(* IEC 61131-3 sources: ecmc_plugin_strucpp/examples/psi_ioc_examples/MTEST04-MTN-STRUCPP/src/generated, 1 file *)

(* ---- main_bundle.st ---- *)
(* Auto-generated by strucpp_bundle_st.py. *)

(* BEGIN ecmc_control.st *)
FUNCTION_BLOCK ECMC_PID
VAR_INPUT
  Enable   : BOOL := TRUE;
  Reset    : BOOL := FALSE;
  Setpoint : LREAL;
  Actual   : LREAL;
  FF       : LREAL := 0.0;
  Kp       : LREAL := 1.0;
  Ki       : LREAL := 0.0;
  Kd       : LREAL := 0.0;
  Kff      : LREAL := 1.0;
  DT       : LREAL := 1.0;
  DFilterTau : LREAL := 0.0;
  OutMin   : LREAL := 0.0;
  OutMax   : LREAL := 0.0;
  IMin     : LREAL := 0.0;
  IMax     : LREAL := 0.0;
END_VAR
VAR_OUTPUT
  Error   : LREAL;
  Output  : LREAL;
  PPart   : LREAL;
  IPart   : LREAL;
  DPart   : LREAL;
  FFPart  : LREAL;
  Limited : BOOL;
END_VAR
VAR
  PrevError    : LREAL;
  DState       : LREAL;
  WasEnabled   : BOOL;
  CandidateI   : LREAL;
  DRaw         : LREAL;
  DAlpha       : LREAL;
  UnsatOutput  : LREAL;
END_VAR

Error := Setpoint - Actual;

IF Reset THEN
  Output := 0.0;
  PPart := 0.0;
  IPart := 0.0;
  DPart := 0.0;
  FFPart := 0.0;
  Limited := FALSE;
  PrevError := Error;
  DState := 0.0;
  WasEnabled := FALSE;
ELSIF NOT Enable THEN
  Error := Setpoint - Actual;
  Output := 0.0;
  PPart := 0.0;
  DPart := 0.0;
  FFPart := FF * Kff;
  Limited := FALSE;
  PrevError := Error;
  DState := 0.0;
  WasEnabled := FALSE;
ELSIF NOT WasEnabled THEN
  PPart := Error * Kp;
  DPart := 0.0;
  FFPart := FF * Kff;
  UnsatOutput := PPart + IPart + FFPart;
  Output := UnsatOutput;
  Limited := FALSE;

  IF OutMax > OutMin THEN
    IF Output > OutMax THEN
      Output := OutMax;
      Limited := TRUE;
    END_IF;
    IF Output < OutMin THEN
      Output := OutMin;
      Limited := TRUE;
    END_IF;
  END_IF;

  PrevError := Error;
  DState := 0.0;
  WasEnabled := TRUE;
ELSE
  PPart := Error * Kp;
  CandidateI := IPart + Error * Ki * DT;

  IF IMax > IMin THEN
    IF CandidateI > IMax THEN
      CandidateI := IMax;
    END_IF;
    IF CandidateI < IMin THEN
      CandidateI := IMin;
    END_IF;
  END_IF;

  IF DT > 0.0 THEN
    DRaw := (Error - PrevError) / DT;
    IF DFilterTau > 0.0 THEN
      DAlpha := DT / (DFilterTau + DT);
      DState := DState + DAlpha * (DRaw - DState);
    ELSE
      DState := DRaw;
    END_IF;
    DPart := Kd * DState;
  ELSE
    DState := 0.0;
    DPart := 0.0;
  END_IF;

  FFPart := FF * Kff;
  UnsatOutput := PPart + CandidateI + DPart + FFPart;
  Output := UnsatOutput;
  Limited := FALSE;

  IF OutMax > OutMin THEN
    IF Output > OutMax THEN
      Output := OutMax;
      Limited := TRUE;
    END_IF;
    IF Output < OutMin THEN
      Output := OutMin;
      Limited := TRUE;
    END_IF;
  END_IF;

  IF (NOT Limited) OR
     ((UnsatOutput > OutMax) AND (Error < 0.0)) OR
     ((UnsatOutput < OutMin) AND (Error > 0.0)) THEN
    IPart := CandidateI;
  END_IF;

  PrevError := Error;
  WasEnabled := TRUE;
END_IF;
END_FUNCTION_BLOCK
(* END ecmc_control.st *)

(* BEGIN ecmc_utils.st *)
FUNCTION_BLOCK ECMC_DebounceBool
VAR_INPUT
  In       : BOOL;
  OnDelay  : TIME := T#0ms;
  OffDelay : TIME := T#0ms;
END_VAR
VAR_OUTPUT
  Out     : BOOL;
  Rising  : BOOL;
  Falling : BOOL;
END_VAR
VAR
  OnTimer  : TON;
  OffTimer : TON;
END_VAR

Rising := FALSE;
Falling := FALSE;

OnTimer(IN := In, PT := OnDelay);
OffTimer(IN := NOT In, PT := OffDelay);

IF In THEN
  IF (OnDelay <= T#0ms) OR OnTimer.Q THEN
    IF NOT Out THEN
      Rising := TRUE;
    END_IF;
    Out := TRUE;
  END_IF;
ELSE
  IF (OffDelay <= T#0ms) OR OffTimer.Q THEN
    IF Out THEN
      Falling := TRUE;
    END_IF;
    Out := FALSE;
  END_IF;
END_IF;
END_FUNCTION_BLOCK

FUNCTION ECMC_ApplyDeadband : LREAL
VAR_INPUT
  Value  : LREAL;
  Width  : LREAL := 0.0;
  Center : LREAL := 0.0;
END_VAR
VAR
  Delta : LREAL;
END_VAR

Delta := Value - Center;
IF Width <= 0.0 THEN
  ECMC_ApplyDeadband := Value;
ELSIF ABS(Delta) <= Width THEN
  ECMC_ApplyDeadband := Center;
ELSIF Delta > 0.0 THEN
  ECMC_ApplyDeadband := Center + (Delta - Width);
ELSE
  ECMC_ApplyDeadband := Center + (Delta + Width);
END_IF;
END_FUNCTION

FUNCTION ECMC_Clamp : LREAL
VAR_INPUT
  Value : LREAL;
  Min   : LREAL := 0.0;
  Max   : LREAL := 0.0;
END_VAR
VAR
  Lo : LREAL;
  Hi : LREAL;
END_VAR

Lo := Min;
Hi := Max;
IF Hi < Lo THEN
  Lo := Max;
  Hi := Min;
END_IF;

IF Hi > Lo THEN
  IF Value < Lo THEN
    ECMC_Clamp := Lo;
  ELSIF Value > Hi THEN
    ECMC_Clamp := Hi;
  ELSE
    ECMC_Clamp := Value;
  END_IF;
ELSE
  ECMC_Clamp := Value;
END_IF;
END_FUNCTION

FUNCTION ECMC_InWindow : BOOL
VAR_INPUT
  Value     : LREAL;
  Low       : LREAL;
  High      : LREAL;
  Inclusive : BOOL := TRUE;
END_VAR
VAR
  Lo : LREAL;
  Hi : LREAL;
END_VAR

Lo := Low;
Hi := High;
IF Hi < Lo THEN
  Lo := High;
  Hi := Low;
END_IF;

IF Inclusive THEN
  ECMC_InWindow := (Value >= Lo) AND (Value <= Hi);
ELSE
  ECMC_InWindow := (Value > Lo) AND (Value < Hi);
END_IF;
END_FUNCTION

FUNCTION ECMC_GetCycleTimeS : LREAL
{external
  extern double ecmcStrucppGetCycleTimeS();
  return ecmcStrucppGetCycleTimeS();
}
END_FUNCTION

FUNCTION_BLOCK ECMC_RateLimiter
VAR_INPUT
  Enable      : BOOL := TRUE;
  Reset       : BOOL := FALSE;
  Input       : LREAL;
  RisingRate  : LREAL := 0.0;
  FallingRate : LREAL := 0.0;
  DT          : LREAL := 1.0;
  InitToInput : BOOL := TRUE;
END_VAR
VAR_OUTPUT
  Output  : LREAL;
  Limited : BOOL;
END_VAR
VAR
  Delta   : LREAL;
  MaxStep : LREAL;
END_VAR

IF Reset OR (NOT Enable) THEN
  IF InitToInput THEN
    Output := Input;
  END_IF;
  Limited := FALSE;
ELSE
  Delta := Input - Output;
  Limited := FALSE;

  IF (DT <= 0.0) THEN
    Output := Input;
  ELSIF Delta > 0.0 THEN
    IF RisingRate <= 0.0 THEN
      Output := Input;
    ELSE
      MaxStep := RisingRate * DT;
      IF Delta > MaxStep THEN
        Output := Output + MaxStep;
        Limited := TRUE;
      ELSE
        Output := Input;
      END_IF;
    END_IF;
  ELSIF Delta < 0.0 THEN
    IF FallingRate <= 0.0 THEN
      Output := Input;
    ELSE
      MaxStep := FallingRate * DT;
      IF (-Delta) > MaxStep THEN
        Output := Output - MaxStep;
        Limited := TRUE;
      ELSE
        Output := Input;
      END_IF;
    END_IF;
  END_IF;
END_IF;
END_FUNCTION_BLOCK

FUNCTION_BLOCK ECMC_FirstOrderFilter
VAR_INPUT
  Enable      : BOOL := TRUE;
  Reset       : BOOL := FALSE;
  Input       : LREAL;
  Tau         : LREAL := 0.0;
  DT          : LREAL := 1.0;
  InitToInput : BOOL := TRUE;
END_VAR
VAR_OUTPUT
  Output : LREAL;
END_VAR
VAR
  Alpha : LREAL;
END_VAR

IF Reset OR (NOT Enable) THEN
  IF InitToInput THEN
    Output := Input;
  END_IF;
ELSIF (Tau <= 0.0) OR (DT <= 0.0) THEN
  Output := Input;
ELSE
  Alpha := DT / (Tau + DT);
  Output := Output + Alpha * (Input - Output);
END_IF;
END_FUNCTION_BLOCK

FUNCTION_BLOCK ECMC_HysteresisBool
VAR_INPUT
  In        : LREAL;
  Low       : LREAL := 0.0;
  High      : LREAL := 0.0;
  Reset     : BOOL := FALSE;
  InitState : BOOL := FALSE;
END_VAR
VAR_OUTPUT
  Out     : BOOL;
  Rising  : BOOL;
  Falling : BOOL;
END_VAR
VAR
  Lo : LREAL;
  Hi : LREAL;
END_VAR

Lo := Low;
Hi := High;
IF Hi < Lo THEN
  Lo := High;
  Hi := Low;
END_IF;

Rising := FALSE;
Falling := FALSE;

IF Reset THEN
  IF Out <> InitState THEN
    Rising := InitState;
    Falling := NOT InitState;
  END_IF;
  Out := InitState;
ELSE
  IF NOT Out THEN
    IF In >= Hi THEN
      Out := TRUE;
      Rising := TRUE;
    END_IF;
  ELSE
    IF In <= Lo THEN
      Out := FALSE;
      Falling := TRUE;
    END_IF;
  END_IF;
END_IF;
END_FUNCTION_BLOCK

FUNCTION_BLOCK ECMC_Integrator
VAR_INPUT
  Enable : BOOL := TRUE;
  Reset  : BOOL := FALSE;
  Hold   : BOOL := FALSE;
  In     : LREAL;
  K      : LREAL := 1.0;
  DT     : LREAL := 1.0;
  Min    : LREAL := 0.0;
  Max    : LREAL := 0.0;
  Init   : LREAL := 0.0;
END_VAR
VAR_OUTPUT
  Out     : LREAL;
  Limited : BOOL;
END_VAR
VAR
  Candidate : LREAL;
  Lo        : LREAL;
  Hi        : LREAL;
END_VAR

Lo := Min;
Hi := Max;
IF Hi < Lo THEN
  Lo := Max;
  Hi := Min;
END_IF;

IF Reset THEN
  Out := Init;
  Limited := FALSE;
ELSIF Enable AND (NOT Hold) AND (DT > 0.0) THEN
  Candidate := Out + In * K * DT;
  Limited := FALSE;

  IF Hi > Lo THEN
    IF Candidate < Lo THEN
      Candidate := Lo;
      Limited := TRUE;
    ELSIF Candidate > Hi THEN
      Candidate := Hi;
      Limited := TRUE;
    END_IF;
  END_IF;

  Out := Candidate;
ELSE
  Limited := FALSE;
END_IF;
END_FUNCTION_BLOCK

FUNCTION_BLOCK ECMC_EcSlaveStatus
VAR_INPUT
  SlaveId  : INT;
  MasterId : INT := -1;
END_VAR
VAR_OUTPUT
  Valid       : BOOL;
  Online      : BOOL;
  Operational : BOOL;
  Init        : BOOL;
  PreOp       : BOOL;
  SafeOp      : BOOL;
  Op          : BOOL;
  StateCode   : BYTE;
  StateWord   : DWORD;
END_VAR
{external
  extern uint32_t ecmcStrucppGetEcSlaveStateWord(int32_t master_index, int32_t slave_index);
  const uint32_t word = ecmcStrucppGetEcSlaveStateWord(MASTERID.get(), SLAVEID.get());
  const uint32_t state_code = (word >> 3u) & 0xFu;

  STATEWORD.set(word);
  STATECODE.set(static_cast<uint8_t>(state_code));
  VALID.set((word & (1u << 0u)) != 0u);
  ONLINE.set((word & (1u << 1u)) != 0u);
  OPERATIONAL.set((word & (1u << 2u)) != 0u);
  INIT.set(state_code == 1u);
  PREOP.set(state_code == 2u);
  SAFEOP.set(state_code == 4u);
  OP.set(state_code == 8u);
}
END_FUNCTION_BLOCK

FUNCTION_BLOCK ECMC_EcMasterStatus
VAR_INPUT
  MasterId : INT := -1;
END_VAR
VAR_OUTPUT
  Valid            : BOOL;
  LinkUp           : BOOL;
  Init             : BOOL;
  PreOp            : BOOL;
  SafeOp           : BOOL;
  Op               : BOOL;
  StateCode        : BYTE;
  SlavesResponding : UINT;
  StateWord        : DWORD;
END_VAR
{external
  extern uint32_t ecmcStrucppGetEcMasterStateWord(int32_t master_index);
  const uint32_t word = ecmcStrucppGetEcMasterStateWord(MASTERID.get());
  const uint32_t state_code = (word >> 2u) & 0xFu;

  STATEWORD.set(word);
  STATECODE.set(static_cast<uint8_t>(state_code));
  VALID.set((word & (1u << 0u)) != 0u);
  LINKUP.set((word & (1u << 1u)) != 0u);
  INIT.set(state_code == 1u);
  PREOP.set(state_code == 2u);
  SAFEOP.set(state_code == 4u);
  OP.set(state_code == 8u);
  SLAVESRESPONDING.set(static_cast<uint16_t>((word >> 16u) & 0xFFFFu));
}
END_FUNCTION_BLOCK

FUNCTION ECMC_AxisGetTrajSource : DINT
VAR_INPUT
  AxisId : DINT;
END_VAR
{external
  extern int32_t ecmcStrucppGetAxisTrajSource(int32_t axis_index);
  return ecmcStrucppGetAxisTrajSource(AXISID.get());
}
END_FUNCTION

FUNCTION ECMC_AxisGetEncSource : DINT
VAR_INPUT
  AxisId : DINT;
END_VAR
{external
  extern int32_t ecmcStrucppGetAxisEncSource(int32_t axis_index);
  return ecmcStrucppGetAxisEncSource(AXISID.get());
}
END_FUNCTION

FUNCTION ECMC_AxisGetActualPos : LREAL
VAR_INPUT
  AxisId : DINT;
END_VAR
{external
  extern double ecmcStrucppGetAxisActualPos(int32_t axis_index);
  return ecmcStrucppGetAxisActualPos(AXISID.get());
}
END_FUNCTION

FUNCTION ECMC_AxisGetSetpointPos : LREAL
VAR_INPUT
  AxisId : DINT;
END_VAR
{external
  extern double ecmcStrucppGetAxisSetpointPos(int32_t axis_index);
  return ecmcStrucppGetAxisSetpointPos(AXISID.get());
}
END_FUNCTION

FUNCTION ECMC_AxisGetActualVel : LREAL
VAR_INPUT
  AxisId : DINT;
END_VAR
{external
  extern double ecmcStrucppGetAxisActualVel(int32_t axis_index);
  return ecmcStrucppGetAxisActualVel(AXISID.get());
}
END_FUNCTION

FUNCTION ECMC_AxisGetSetpointVel : LREAL
VAR_INPUT
  AxisId : DINT;
END_VAR
{external
  extern double ecmcStrucppGetAxisSetpointVel(int32_t axis_index);
  return ecmcStrucppGetAxisSetpointVel(AXISID.get());
}
END_FUNCTION

FUNCTION ECMC_AxisIsEnabled : BOOL
VAR_INPUT
  AxisId : DINT;
END_VAR
{external
  extern int32_t ecmcStrucppGetAxisEnabled(int32_t axis_index);
  return ecmcStrucppGetAxisEnabled(AXISID.get()) != 0;
}
END_FUNCTION

FUNCTION ECMC_AxisIsBusy : BOOL
VAR_INPUT
  AxisId : DINT;
END_VAR
{external
  extern int32_t ecmcStrucppGetAxisBusy(int32_t axis_index);
  return ecmcStrucppGetAxisBusy(AXISID.get()) != 0;
}
END_FUNCTION

FUNCTION ECMC_AxisHasError : BOOL
VAR_INPUT
  AxisId : DINT;
END_VAR
{external
  extern int32_t ecmcStrucppGetAxisError(int32_t axis_index);
  return ecmcStrucppGetAxisError(AXISID.get()) != 0;
}
END_FUNCTION

FUNCTION ECMC_AxisGetErrorId : DINT
VAR_INPUT
  AxisId : DINT;
END_VAR
{external
  extern int32_t ecmcStrucppGetAxisErrorId(int32_t axis_index);
  return ecmcStrucppGetAxisErrorId(AXISID.get());
}
END_FUNCTION

FUNCTION ECMC_AxisSetTrajSource : DINT
VAR_INPUT
  AxisId : DINT;
  Source : DINT;
END_VAR
{external
  extern int32_t ecmcStrucppSetAxisTrajSource(int32_t axis_index, int32_t source);
  return ecmcStrucppSetAxisTrajSource(AXISID.get(), SOURCE.get());
}
END_FUNCTION

FUNCTION ECMC_AxisSetEncSource : DINT
VAR_INPUT
  AxisId : DINT;
  Source : DINT;
END_VAR
{external
  extern int32_t ecmcStrucppSetAxisEncSource(int32_t axis_index, int32_t source);
  return ecmcStrucppSetAxisEncSource(AXISID.get(), SOURCE.get());
}
END_FUNCTION

FUNCTION ECMC_AxisUseInternalTraj : DINT
VAR_INPUT
  AxisId : DINT;
END_VAR
  ECMC_AxisUseInternalTraj := ECMC_AxisSetTrajSource(AxisId := AxisId, Source := 0);
END_FUNCTION

FUNCTION ECMC_AxisUseExternalTraj : DINT
VAR_INPUT
  AxisId : DINT;
END_VAR
  ECMC_AxisUseExternalTraj := ECMC_AxisSetTrajSource(AxisId := AxisId, Source := 1);
END_FUNCTION

FUNCTION ECMC_AxisUseInternalEnc : DINT
VAR_INPUT
  AxisId : DINT;
END_VAR
  ECMC_AxisUseInternalEnc := ECMC_AxisSetEncSource(AxisId := AxisId, Source := 0);
END_FUNCTION

FUNCTION ECMC_AxisUseExternalEnc : DINT
VAR_INPUT
  AxisId : DINT;
END_VAR
  ECMC_AxisUseExternalEnc := ECMC_AxisSetEncSource(AxisId := AxisId, Source := 1);
END_FUNCTION

FUNCTION ECMC_AxisSetExternalSetpointPos : DINT
VAR_INPUT
  AxisId   : DINT;
  Position : LREAL;
END_VAR
{external
  extern int32_t ecmcStrucppSetAxisExtSetPos(int32_t axis_index, double value);
  return ecmcStrucppSetAxisExtSetPos(AXISID.get(), POSITION.get());
}
END_FUNCTION

FUNCTION ECMC_AxisSetExternalEncoderPos : DINT
VAR_INPUT
  AxisId   : DINT;
  Position : LREAL;
END_VAR
{external
  extern int32_t ecmcStrucppSetAxisExtActPos(int32_t axis_index, double value);
  return ecmcStrucppSetAxisExtActPos(AXISID.get(), POSITION.get());
}
END_FUNCTION
(* END ecmc_utils.st *)

(* BEGIN ecmc_debug.st *)
FUNCTION_BLOCK ECMC_DebugPrint
VAR_INPUT
  Execute : BOOL;
  Message : STRING;
END_VAR
VAR_OUTPUT
  Fired : BOOL;
END_VAR
VAR
  PrevExecute : BOOL;
END_VAR
{external
  const bool execute = EXECUTE.get();
  FIRED.set(false);

  if (execute && !PREVEXECUTE.get()) {
    const auto message = MESSAGE.get();
    extern void ecmcStrucppDebugPrint(const char* message);
    ecmcStrucppDebugPrint(message.c_str());
    FIRED.set(true);
  }

  PREVEXECUTE.set(execute);
}
END_FUNCTION_BLOCK

FUNCTION ECMC_DebugPrintNow : BOOL
VAR_INPUT
  Message : STRING;
END_VAR
{external
  const auto message = MESSAGE.get();
  extern void ecmcStrucppDebugPrint(const char* message);
  ecmcStrucppDebugPrint(message.c_str());
  return true;
}
END_FUNCTION
(* END ecmc_debug.st *)

(* BEGIN main.st *)
PROGRAM MAIN
VAR
  actual_position    AT %IW0 : INT;   // @ecmc ec.s14.positionActual01
  drive_control      AT %QW0 : WORD;  // @ecmc ec.s14.driveControl01
  velocity_setpoint  AT %QW2 : INT;   // @ecmc ec.s14.velocitySetpoint01
  cycle_counter      AT %MW0 : INT;   // @epics rec=Main-CycleCounterAct
  actual_pos_export          : INT;   // @epics prefix=$(IOC): rec=Main-PosActMini
  dbg_sample_trigger         : BOOL;
  startup_printed            : BOOL;
  dbg_startup                : ECMC_DebugPrint;
  dbg_position               : ECMC_DebugPrint;
  dbg_reverse_pos            : ECMC_DebugPrint;
  dbg_reverse_neg            : ECMC_DebugPrint;
END_VAR

actual_pos_export := actual_position;
cycle_counter := cycle_counter + 1;
drive_control := 16#0001;

dbg_startup(Execute := NOT startup_printed,
            Message := 'ST program started');
startup_printed := TRUE;

dbg_sample_trigger := (cycle_counter MOD 1000) = 0;
dbg_position(Execute := dbg_sample_trigger,
             Message := CONCAT('actual_position=',
                               TO_STRING(actual_position)));

IF velocity_setpoint = 0 THEN
  velocity_setpoint := 1000;
END_IF;

IF actual_position <= 0 THEN
  velocity_setpoint := 1000;
ELSIF actual_position >= 12800 THEN
  velocity_setpoint := -1000;
END_IF;

dbg_reverse_pos(Execute := actual_position <= 0,
                Message := CONCAT('reverse -> +1000 at pos=',
                                  TO_STRING(actual_position)));
dbg_reverse_neg(Execute := actual_position >= 12800,
                Message := CONCAT('reverse -> -1000 at pos=',
                                  TO_STRING(actual_position)));
END_PROGRAM
(* END main.st *)
